// TwinCAT 3 PLC project Device
// ProgramVersion: 3.1.4024.0
// libraries:
//   Tc2_Standard, * (Beckhoff Automation GmbH)
//   Tc2_System, * (Beckhoff Automation GmbH)
//   Tc2_Utilities, * (Beckhoff Automation GmbH)
//   Tc3_IotBase, * (Beckhoff Automation GmbH)
//   Tc3_JsonXml, * (Beckhoff Automation GmbH)
//   Tc3_Module, * (Beckhoff Automation GmbH)
// project tree:
//   DUTs/ DeviceAttr.TcDUT
//   GVLs/ GVL.TcGVL
//   / PlcTask.TcTTO
//   POUs/ DIGIIOT_UPDATE.TcPOU, FB_EventHTTP_Post.TcPOU, FB_UpdateTimeStamp.TcPOU, MAIN.TcPOU, MSG_CONCAT.TcPOU, FB_UnixTimestamp.TcPOU
// real-time tasks:
//   TASK PlcTask: cycle T#10ms, priority 20, ADS port 350

CONFIGURATION Device
    RESOURCE PLC ON TwinCAT3
        TASK PlcTask(INTERVAL := T#10ms, PRIORITY := 20);
        PROGRAM MAIN WITH PlcTask : MAIN;
    END_RESOURCE
END_CONFIGURATION

// ---- DUTs/DeviceAttr.TcDUT
TYPE DeviceAttr :
STRUCT
	DeviceID : STRING(40);
	ActionKey : STRING(20);
	ActionVal : USINT;
	OnlineKey : STRING(6) := 'Online';
	OnlineVal : USINT;
	ErrorKey  : STRING(5) := 'Error';
	ErrorVal  : USINT;
END_STRUCT
END_TYPE

// ---- GVLs/GVL.TcGVL
{attribute 'qualified_only'}
VAR_GLOBAL
	API_MSG : STRING(3500);
END_VAR

// ---- POUs/MAIN.TcPOU
PROGRAM MAIN
VAR
	
//	IPAdress		: STRING 	:= '192.168.1.132';
//	Port			: UINT		:= 5000;
	IPAdress		: STRING 	:= '10.0.110.19';
	Port			: UINT		:= 6060;
	UpdatePeriod	: TIME		:= T#60S;
	Timer 			: BOOL;
	
	API_MSG			: STRING(3500);
	HttpSend		: BOOL := FALSE;
	bSuccess		: BOOL;
	bError			: BOOL;
	
	fb_TimeStamp	: FB_UpdateTimeStamp;
	fb_httppost		: FB_EventHTTP_Post;
	fbTON 	: TON;
	fbTOFF 	: TON;
	Rise1	: R_TRIG;
	
	fbHttpProcess	: FB_IotHttpClient :=(	sHostName			:= IPAdress,
								  			bKeepAlive			:= TRUE, 
											tConnectionTimeout	:= T#10S);
	enabler	: bool;
END_VAR


IF NOT fbHttpProcess.bConfigured THEN 
	fbHttpProcess.nHostPort 				:= Port;
	fbHttpProcess.stTLS.bNoServerCertCheck 	:= FALSE;
END_IF
	
fb_TimeStamp();
IF fb_TimeStamp.timeValid THEN
		
//	fbTON(IN := NOT fbTOFF.Q, PT := T#0.5S);
//	fbTOFF (IN := fbTON.Q, PT := T#0.5S);

//	Rise1(CLK:=fbTON.Q);

	Rise1(CLK:= enabler);
	IF Rise1.Q THEN
		HttpSend := TRUE;
		DIGIIOT_UPDATE(SystemTime := fb_TimeStamp.timestampSeconds);
	END_IF
	
	IF fbHttpProcess.bConfigured THEN 
		fb_httppost( 	bSend		:= HttpSend, 
						fbClient	:= fbHttpProcess, 
						API_URI		:= '/upload',
//						API_Msg 	:= '{"station": 1, "start_ts": "2025-01-24 13:30:00", "end_ts": "2025-01-24 13:31:00"}',
						API_Msg		:= GVL.API_MSG,
						bSuccess 	=> bSuccess,
						bError		=> bError );
						
		IF fb_httppost.bSuccess OR fb_httppost.bError THEN
			HttpSend := FALSE;
		END_IF
	END_IF 
	fbHttpProcess.Execute();
END_IF

END_PROGRAM

// ---- POUs/FB_UpdateTimeStamp.TcPOU
FUNCTION_BLOCK FB_UpdateTimeStamp
VAR_INPUT
END_VAR
VAR_OUTPUT
	FullSystemTime	: STRING;
	SystemDate		: STRING;
	SystemTime		: STRING;
	SystemHour		: STRING;
	timeValid		: BOOL;
    timestampSeconds: STRING;
END_VAR
VAR
	fb_LocalTime	 : FB_LocalSystemTime;
    stLocalTime : TIMESTRUCT;  
	unixTime: FB_UnixTimestamp;
END_VAR

fb_LocalTime(
		sNetID:= , 
		bEnable:= TRUE , 
		dwCycle:= 1, 
		dwOpt:= , 
		tTimeout:= ,
		bValid=> timeValid, 
		systemTime=> stLocalTime, 
		tzID=> );
		
IF fb_localTime.bValid THEN
//	FullSystemTime 	:= SYSTEMTIME_TO_STRING(fb_LocalTime.systemTime);
	
//	SystemDate		:= WORD_TO_STRING(fb_LocalTime.systemTime.wYear);
//	SystemDate		:= CONCAT(SystemDate, '.');
//	SystemDate		:= CONCAT(SystemDate, WORD_TO_STRING(fb_LocalTime.systemTime.wMonth));
//	SystemDate		:= CONCAT(SystemDate, '.');
//	SystemDate		:= CONCAT(SystemDate, WORD_TO_STRING(fb_LocalTime.systemTime.wDay));
	
//	SystemTime		:= WORD_TO_STRING(fb_LocalTime.systemTime.wHour);
//	SystemTime		:= CONCAT(SystemTime, ':');
//	SystemTime		:= CONCAT(SystemTime, WORD_TO_STRING(fb_LocalTime.systemTime.wMinute));
//	SystemTime		:= CONCAT(SystemTime, ':');
//	SystemTime		:= CONCAT(SystemTime, WORD_TO_STRING(fb_LocalTime.systemTime.wSecond));
	
//	SystemHour		:= WORD_TO_STRING(fb_LocalTime.systemTime.wHour);
	
	unixTime();
	timestampSeconds := ULINT_TO_STRING(unixTime.seconds);
END_IF

END_FUNCTION_BLOCK

// ---- POUs/FB_UnixTimestamp.TcPOU
FUNCTION_BLOCK FB_UnixTimestamp
VAR_OUTPUT
    seconds: ULINT;
//    milliseconds: ULINT;
END_VAR

VAR
    localSystemTime : FB_LocalSystemTime := ( bEnable := TRUE, dwCycle := 1 );
    getTimeZoneInformation : FB_GetTimeZoneInformation;
    timeZoneInformation : ST_TimeZoneInformation;
    specificLocalTimeToFileTime : FB_TzSpecificLocalTimeToFileTime;
    fileTime: T_FILETIME;
    onZerothSecondLastCycle : BOOL;
END_VAR

// Get local system time
localSystemTime();

// On the zeroth second of each minutesync timezone information
IF (timeZoneInformation.standardName = '' OR (localSystemTime.systemTime.wSecond = 0 AND NOT onZerothSecondLastCycle)) THEN
    getTimeZoneInformation(sNetID := '', bExecute := TRUE, tzInfo => timeZoneInformation);
END_IF;

// Convert local system time to unix timestamps
specificLocalTimeToFileTime(in := Tc2_Utilities.SYSTEMTIME_TO_FILETIME(localSystemTime.systemTime), tzInfo := timeZoneInformation, out => fileTime);
seconds := (SHL(DWORD_TO_ULINT(fileTime.dwHighDateTime), 32) + DWORD_TO_ULINT(fileTime.dwLowDateTime)) / 10000000 - 11644473600;
//milliseconds := (SHL(DWORD_TO_ULINT(fileTime.dwHighDateTime), 32) + DWORD_TO_ULINT(fileTime.dwLowDateTime)) / 10000 - 11644473600000;

onZerothSecondLastCycle := localSystemTime.systemTime.wSecond = 0;

END_FUNCTION_BLOCK

// ---- POUs/FB_EventHTTP_Post.TcPOU
FUNCTION_BLOCK FB_EventHTTP_Post
VAR_INPUT
	bSend		: BOOL;
	API_URI		: STRING[255];
	API_Msg		: STRING[3500];
END_VAR
VAR_IN_OUT
	fbClient			: FB_IotHttpClient;
END_VAR
VAR_OUTPUT
	bSuccess			: Bool;
	bBusy				: BOOL;
	bError				: BOOL;
END_VAR
VAR	
	// set content to json
	API_STR     		: STRING(Tc3_IotBase.ParameterList.cSizeOfHttpContentType-1) := 'application/json';

	fbRequest			: FB_IotHttpRequest;
	fbHeader			: FB_IotHttpHeaderFieldMap;
	fbJson				: FB_JsonDomParser;
	
 	dtTimestamp    		: DATE_AND_TIME := DT#2017-04-04-12:42:42;
	fbJsonWriter		: FB_JsonDomParser;
	nState				: UDINT;
	RisingEdge			: R_TRIG;
	
	bGetContentResult	: BOOL;
	sContent			: STRING[5000] := ''; 
	
	bGetJsonResult		: BOOL;
	jsonDoc				: SJsonValue;
	jsonVal				: SJsonValue;
	sResultValue		: STRING;
	sResultValue2		: STRING;
	bOnce				: BOOL := TRUE;
	
	nReqCount			: UDINT;
	nResCount			: UDINT;
	nValidResCount		: UDINT;
	nErrCount			: UDINT;	
END_VAR

RisingEdge(CLK:= bSend);
IF bOnce THEN
	fbHeader.AddField('x-api-key', '8e0697a446bd2c17b4e1188f1d21439ef863aa79b59e31981a7135b3171f9b85', FALSE);	
	bOnce:= FALSE;
END_IF
CASE nState OF
0:		
	IF RisingEdge.Q THEN 
		sContent := API_Msg;
		fbRequest.sContentType := API_STR;
		IF fbRequest.SendRequest(sUri:= API_URI, fbClient:= fbClient, eRequestType:= ETcIotHttpRequestType.HTTP_POST, pContent:= ADR(sContent), nContentSize:= LEN2(ADR(sContent)), fbHeader) THEN				
			nState:= 1;
			bBusy:= TRUE;
			bError:= FALSE;
			bSuccess := FALSE;
		END_IF					
	END_IF
1:
	IF NOT fbRequest.bBusy THEN
		bError:= TRUE;
		IF NOT fbRequest.bError THEN
							 				
			bGetContentResult:= fbRequest.GetContent(pContent:= ADR(sContent), nContentSize:= SIZEOF(SContent), bSetNullTermination:= TRUE);	
			IF fbRequest.nStatusCode >= 200 AND fbRequest.nStatusCode < 300 THEN
				bGetJsonResult:= FALSE;
//				jsonDoc:= fbRequest.GetJsonDomContent(fbJson);				
//				IF jsonDoc <> 0 THEN
//					bGetJsonResult:= TRUE;
//					IF fbJson.HasMember(jsonDoc, 'status')  THEN
//						jsonVal:= fbJson.FindMember(jsonDoc, 'status');	
//						sResultValue:= fbJson.GetString(jsonVal);
//						IF sResultValue = 'success' THEN
							nValidResCount:= nValidResCount+1;	
							bSuccess := TRUE;
							bError:= FALSE;
//						END_IF
//					END_IF		
//				END_IF
				nResCount:= nResCount+1;					
			END_IF				
		END_IF
		nState:= 0;
		bBusy:= FALSE;
		IF bError THEN
			nErrCount:= nErrCount+1;
		END_IF		
	END_IF 
END_CASE

END_FUNCTION_BLOCK

// ---- POUs/DIGIIOT_UPDATE.TcPOU
PROGRAM DIGIIOT_UPDATE
VAR_INPUT
	SystemTime : STRING;
END_VAR
VAR
	DeviceState : ARRAY[1..14] OF DeviceAttr;
	KR_Action	: ARRAY[1..14] OF STRING;
	KR_Error	: ARRAY[1..14] OF USINT;
	KR_Online	: ARRAY[1..14] OF USINT;
	
	index : INT;
	API_MSG : STRING(3500);
END_VAR


DeviceState[1].DeviceID := 'WC1_KR1';
DeviceState[1].ActionKey := 'JigBToTTorch';
DeviceState[2].DeviceID := 'WC1_KR2';
DeviceState[2].ActionKey := 'WeldJigB';
DeviceState[3].DeviceID := 'WC1_KR3';
DeviceState[3].ActionKey := 'PlaceJigCTo_CR01';
DeviceState[4].DeviceID := 'WC1_KR4';
DeviceState[4].ActionKey := 'WeldJigC';
DeviceState[5].DeviceID := 'WC1_KR5';
DeviceState[5].ActionKey := 'COSMOToConveyor';
DeviceState[6].DeviceID := 'WC1_INFEEDRACK';
DeviceState[6].ActionKey := 'Sensor_A5';
DeviceState[7].DeviceID := 'WC1_JIGA';
DeviceState[7].ActionKey := 'Clamp';
DeviceState[8].DeviceID := 'WC1_JIGB';
DeviceState[8].ActionKey := 'Clamp';
DeviceState[9].DeviceID := 'WC1_JIGC';
DeviceState[9].ActionKey := 'Clamp';
DeviceState[10].DeviceID := 'WC1_TWINTORCH';
DeviceState[10].ActionKey := 'Run';
DeviceState[11].DeviceID := 'WC1_COSMOS_LEAK_TESTER';
DeviceState[11].ActionKey := 'Run';
DeviceState[12].DeviceID := 'WC1_REWORK_JIG_Conveyor';
DeviceState[12].ActionKey := 'ConveyorFull';
DeviceState[13].DeviceID := 'WC1_COOLINGRACK';
DeviceState[13].ActionKey := 'CR01';
DeviceState[14].DeviceID := 'WC1_VibratorBowl';
DeviceState[14].ActionKey := 'VB_Ready';

FOR index:=1 TO 2 DO 
	DeviceState[index].OnlineVal := KR_Online[index];
	DeviceState[index].OnlineVal := KR_Error[index];
END_FOR

API_MSG := MSG_CONCAT(_DeviceState := DeviceState, _SystemTime := SystemTime);
GVL.API_MSG := API_MSG;

END_PROGRAM

// ---- POUs/MSG_CONCAT.TcPOU
FUNCTION MSG_CONCAT : STRING(3500)
VAR_INPUT
	_DeviceState : ARRAY[1..14] OF DeviceAttr;
	_SystemTime	 : STRING;
END_VAR
VAR
	API_JSON		: ARRAY[1..14] OF STRING(255);
	index			: INT;
	success			: BOOL;
	API_MSG			: STRING(3500);
	sopenBracket	: STRING(13) := '{"dbLists":[';
END_VAR


//success := CONCAT2(pSrcString1 := ADR(_text), pSrcString2 := ADR(_SystemTime), pDstString := ADR(API_JSON), nDstSize := SIZEOF(API_JSON));

FOR index:=1 TO 14 DO 
	API_JSON[index] := CONCAT(API_JSON[index],'{"ObjectData":{"ObjectId":"');	
	API_JSON[index] := CONCAT(API_JSON[index],_DeviceState[index].DeviceID);
	API_JSON[index] := CONCAT(API_JSON[index],'","ActionData":[{"Key":"');
	API_JSON[index] := CONCAT(API_JSON[index],_DeviceState[index].ActionKey);
	API_JSON[index] := CONCAT(API_JSON[index],'","Value":"');
	API_JSON[index] := CONCAT(API_JSON[index],USINT_TO_STRING(_DeviceState[index].ActionVal));
	API_JSON[index] := CONCAT(API_JSON[index],'","TimeStamp":');
	API_JSON[index] := CONCAT(API_JSON[index],_SystemTime);
	API_JSON[index] := CONCAT(API_JSON[index],'}],"Attributes":[{"Key":"');
	API_JSON[index] := CONCAT(API_JSON[index],_DeviceState[index].OnlineKey);
	API_JSON[index] := CONCAT(API_JSON[index],'","Value":"');
	API_JSON[index] := CONCAT(API_JSON[index],USINT_TO_STRING(_DeviceState[index].OnlineVal));
	API_JSON[index] := CONCAT(API_JSON[index],'","TimeStamp":');
	API_JSON[index] := CONCAT(API_JSON[index],_SystemTime);
	API_JSON[index] := CONCAT(API_JSON[index],'},{"Key":"');
	API_JSON[index] := CONCAT(API_JSON[index],_DeviceState[index].ErrorKey);
	API_JSON[index] := CONCAT(API_JSON[index],'","Value":"');
	API_JSON[index] := CONCAT(API_JSON[index],USINT_TO_STRING(_DeviceState[index].ErrorVal));
	API_JSON[index] := CONCAT(API_JSON[index],'","TimeStamp":');
	API_JSON[index] := CONCAT(API_JSON[index],_SystemTime);
	IF index < 14 THEN
		API_JSON[index] := CONCAT(API_JSON[index],'}]}},');
	ELSE
		API_JSON[index] := CONCAT(API_JSON[index],'}]}}]}');
	END_IF
	success := CONCAT2(pSrcString1 := ADR(API_MSG), pSrcString2 := ADR(API_JSON[index]), pDstString := ADR(API_MSG), nDstSize := SIZEOF(API_MSG));
END_FOR
	success := CONCAT2(pSrcString1 := ADR(sopenBracket), pSrcString2 := ADR(API_MSG), pDstString := ADR(API_MSG), nDstSize := SIZEOF(API_MSG));
MSG_CONCAT := API_MSG;

END_FUNCTION
